(* PLC project DCCM_PCL_2, Machine Expert Logic Builder V20.2.8.0, author jrfsc *)
(* stored: creationDateTime 2022-12-21T11:20:35.1707039, version 0.0.0.0, modificationDateTime 2022-12-21T11:18:43.8929083 *)

{attribute 'qualified_only'}
VAR_GLOBAL  (* DCCMNVL *)
  RM1_ISO_MODE AT %MW9000 : INT;
  RM2_ISO_MODE AT %MW9001 : INT;
  RM3_ISO_MODE AT %MW9002 : INT;
  RM4_ISO_MODE AT %MW9003 : INT;
END_VAR
